// TIA Portal V20 export
// export: Created 2025-12-01T14:57:44.9159736Z, ExportSetting None, DisplayName Totally Integrated Automation Portal, DisplayVersion V20 Update 3, DisplayName TIA Portal Openness, DisplayVersion V20 Update 3, DisplayName TIA Portal Version Control Interface, DisplayVersion V20 Update 3, DisplayName STEP 7 Professional, DisplayVersion V20 Update 3, DisplayName STEP 7 Safety, DisplayVersion V20 Update 2, DisplayName WinCC Basic/Comfort/Advanced, DisplayVersion V20 Update 3, DisplayName WinCC Professional, DisplayVersion V20 Update 3, DisplayName WinCC Unified, DisplayVersion V20 Update 3
FUNCTION "FC780_Evento_RUET" : Void   // FC780, LAD
{ S7_Optimized_Access := 'FALSE' }
// stored: AutoNumber false, SetENOAutomatically false
   VAR_INPUT
      mensaje : Int;   // indice del array que estamos extrayendo
   END_VAR
   VAR_TEMP
      Existe_ruta : Bool;
      retval : Int;
      pos_SSCC : UInt;
      cero : Byte;
      destinos : Array[0..9] of UInt;
      registro_etiqueta : "ROUT_Reg_Etiqueta";
      orden_desvio : Byte;
      desvio_bits AT orden_desvio : Array[1..8] of Bool;
      posicion : Int;
      pos_ruta : Int;
      posicion_mesa : Int;
      posicion_db : Int;
      desvio : Int;
      scanner : UInt;
      bit_ini : Int;
      n_bits : Int;
      contador_aux : Int;
      contador : Int;
      posicion_BBDD : UInt;
      pos_DB : UInt;
      posicion_libre_BBDD : UInt;
      cola : UInt;
      mi_siguiente : UInt;
      dato_actual_cola : UInt;
   END_VAR
BEGIN

REGION Network 1 (SCL): INICIALIZACIONES
   REGION inicializacion

       // inicializamos las variables
       // 
       #cero := 0;
       #retval := FILL(BVAL := #cero, BLK => #registro_etiqueta); // el registro de la etiqueta temporal
       #retval := FILL(BVAL := #cero, BLK => #destinos); // los datos temporales de los destinos
       #orden_desvio := 0;
       #Existe_ruta := false;
       #pos_SSCC := 0;

   END_REGION
END_REGION

REGION Network 2 (SCL): RECOJO Y CONVIERTO EL VALOR DE LA EITQUETA
   // buscamos donde empieza el SSCC en el mensaje y lo convertimos
   // 
   #pos_SSCC := FIND(IN1 := "DB199_eventos_convertidos".evento[#mensaje], IN2 := '[SSCC]');

   STRG_VAL(IN := "DB199_eventos_convertidos".evento[#mensaje],
            FORMAT := 0,
            P := (#pos_SSCC + 6), // +6 por lo que ocupa el atributo ['SSCC]'
            OUT => #registro_etiqueta.CDB);
END_REGION

REGION Network 3 (SCL): EXTRAEMOS DEL MENSAJE LOS DESTINOS

   // miramos si en el mensaje nos han llegado destinos que extraer
   #posicion := FIND(IN1 := "DB199_eventos_convertidos".evento[#mensaje], IN2 := '[DEST]');
   IF #posicion <> 0 THEN    // iniciamos la estracción de las mesas que pertenecen a la ruta
           // si solamente se ejecuta el proceso una vez en el mensaje no es necesario realizar esta operación de sustituir el atributo DEST
       "DB199_eventos_convertidos".evento[#mensaje] := REPLACE(IN1 := "DB199_eventos_convertidos".evento[#mensaje], IN2 := '[dest]', L := 6, P := #posicion);
       #pos_ruta := 0;
       #Existe_ruta := 1;
       // temporalmente ponemos las rutas a cero
       WHILE #Existe_ruta DO
           #posicion := FIND(IN1 := "DB199_eventos_convertidos".evento[#mensaje], IN2 := '[MESA]');
           IF #posicion <> 0 THEN
               STRG_VAL(IN := "DB199_eventos_convertidos".evento[#mensaje],
                        FORMAT := 0,
                        P := (#posicion + 6),
                        OUT => #destinos[#pos_ruta]);
               #pos_ruta += 1; // incrementamos la posición en el array para seguir guardando
               // las mesas ya extraidas, las ponemos en minucula para seguir buscando las siguientes mesas sin eliminar parcialmente el mensaje
               "DB199_eventos_convertidos".evento[#mensaje] := REPLACE(IN1 := "DB199_eventos_convertidos".evento[#mensaje], IN2 := '[mesa]', L := 6, P := #posicion);
           ELSE
               #Existe_ruta := 0;
               EXIT;
           END_IF;
       END_WHILE;
   END_IF;
   // aqui tenemos que incluir la conversión de las mesas el los bits de cruce
END_REGION

REGION Network 4 (SCL): generamos los bits de cruce
   REGION generar_bits_cruce
       #posicion_mesa := 0;
       #posicion_db := 0;

       WHILE #destinos[#posicion_mesa] <> 0 DO
           // Statement section WHILE

           WHILE (("DB913_Router_DestinoDesvio".DestinoDesvios[#posicion_db].Destino <> 0) AND (#posicion_db <= "ROUT_Max_Destinos")) DO
               IF (#destinos[#posicion_mesa] = "DB913_Router_DestinoDesvio".DestinoDesvios[#posicion_db].Destino) THEN
                   // si coincide la mesa con uno de los destinos
                   #desvio := 0;
                   WHILE (("DB913_Router_DestinoDesvio".DestinoDesvios[#posicion_db].Desvios[#desvio].SCR <> 0) AND (#desvio <= "ROUT_Max_Destinos")) DO
                       #scanner := "DB913_Router_DestinoDesvio".DestinoDesvios[#posicion_db].Desvios[#desvio].SCR;
                       #orden_desvio := "DB913_Router_DestinoDesvio".DestinoDesvios[#posicion_db].Desvios[#desvio].Bits;
                       #bit_ini := "DB912_Tipo_Scanner_Router".SCANNER[#scanner].Bit_Ini_Ordenes;
                       #n_bits := "DB912_Tipo_Scanner_Router".SCANNER[#scanner].N_Bits_Orden;

                       // aqui mediante un for vamos escribiendo los bits donde corresponden
                       #contador_aux := 1;
                       FOR #contador := #bit_ini TO (#bit_ini + #n_bits - 1) DO
                           #registro_etiqueta.BIT_Orden[#contador] := #desvio_bits[#contador_aux];
                           #contador_aux += 1;

                       END_FOR;
                       #desvio += 1; // nos desplazamos el siguiente desvio
                   END_WHILE;

               END_IF;
               #posicion_db += 1; //nos desplazamos hasta el siguiente destino
           END_WHILE;
           #posicion_mesa += 1; // nos desplazamos a la siguiente mesa destino de la ruta
           #posicion_db := 0; // inicializamos a cero la busqueda dentro del DB de destinos

       END_WHILE;

   END_REGION
END_REGION

REGION Network 5 (SCL)
   // ahora que tenemos todos los datos, tenemos que guardarlos.
   // miramos si la etiqueta ya está dada de alta en la BBDD
   // 

   "FC715_Router_BuscarEtiqueta_Lint"(Etiqueta := #registro_etiqueta.CDB,
                                      Posicion_BBDD => #posicion_BBDD);

   // si nos da una posición dentro de la BBDD lo unico que tenemos que hacer es sobreescribir el registo
   // si nos da cero, es que no existe y hay que crearla en la primera posición que esté libre
   // 

   REGION escribir_etiqueta_en_BBDD
       // la etiqueta existe
       // 

       REGION existe_etiqueta
           IF #posicion_BBDD <> 0 THEN
               // en función de la posición que nos devuelva, tenemos que ir a un DB diferente
               // 
               REGION elegir_db_busqueda
                   CASE #posicion_BBDD OF
                       1..1000:
                           #pos_DB := #posicion_BBDD;
                           "DB201_RegEtiquetas_0001_1000".Reg_Etiqueta[#pos_DB].BIT_Orden := #registro_etiqueta.BIT_Orden;
                       1001..2000:
                           #pos_DB := #posicion_BBDD - 1000;
                           "DB202_RegEtiquetas_1001_2000".Reg_Etiqueta[#pos_DB].BIT_Orden := #registro_etiqueta.BIT_Orden;

                       2001..3000:
                           #pos_DB := #posicion_BBDD - 2000;
                           "DB203_RegEtiquetas_2001_3000".Reg_Etiqueta[#pos_DB].BIT_Orden := #registro_etiqueta.BIT_Orden;
                       3001..4000:
                           #pos_DB := #posicion_BBDD - 3000;
                           "DB204_RegEtiquetas_3001_4000".Reg_Etiqueta[#pos_DB].BIT_Orden := #registro_etiqueta.BIT_Orden;
                       ELSE
                           #posicion_BBDD := 0;
                           RETURN;
                   END_CASE;
               END_REGION


               ;
           END_IF;
       END_REGION


       REGION no_existe_etiqueta
           IF #posicion_BBDD = 0 THEN
               // 
               // buscamos la primera posición libre dentro de la BBDD que es lo mismo que buscar la primera etiqueta 0
               // 
               "FC715_Router_BuscarEtiqueta_Lint"(Etiqueta := -1,
                                                  Posicion_BBDD => #posicion_libre_BBDD);

               // si la posicion que devuelve es -1 no hay sitio en la BBDD y no se puede crear la etiqueta.
               // 

               IF #posicion_libre_BBDD = -1 THEN
                   "FC818_Mensaje_BBDD_Routing_Llena"(Etiqueta:=#registro_etiqueta.CDB,
                                                      Envio_JDT2:=(NOT("ROUT_X_CONEX_JDT1")));
                   RETURN;

               END_IF;


               // tambien vamos a extraer el valor de la primera etiqueta de la cola para mantener la coherencia de las colas
               // 
               #cola := #registro_etiqueta.CDB MOD "ROUT_N_Colas";
               #dato_actual_cola := "DB212_Cola_Activa".Cola[#cola];
               "DB212_Cola_Activa".Cola[#cola] := #posicion_libre_BBDD;

               IF #dato_actual_cola <> 0 THEN
                   // no es la primera etiqueta de la cola
                   // ahora yo seré el primero de la cola, y el indicado por el valor dato actual será mi siguiente
                   // y yo su anterior
                   // 



                   CASE #dato_actual_cola OF
                       1..1000:
                           #pos_DB := #dato_actual_cola;
                           "DB201_RegEtiquetas_0001_1000".Reg_Etiqueta[#pos_DB].Anterior := #posicion_libre_BBDD;

                       1001..2000:
                           #pos_DB := #dato_actual_cola - 1000;
                           "DB202_RegEtiquetas_1001_2000".Reg_Etiqueta[#pos_DB].Anterior := #posicion_libre_BBDD;

                       2001..3000:
                           #pos_DB := #dato_actual_cola - 2000;
                           "DB203_RegEtiquetas_2001_3000".Reg_Etiqueta[#pos_DB].Anterior := #posicion_libre_BBDD;
                       3001..4000:
                           #pos_DB := #dato_actual_cola - 3000;
                           "DB204_RegEtiquetas_3001_4000".Reg_Etiqueta[#pos_DB].Anterior := #posicion_libre_BBDD;

                           RETURN;
                   END_CASE;

                   #registro_etiqueta.Posterior := #dato_actual_cola;
               END_IF;

               REGION elegir_db_busqueda
                   CASE #posicion_libre_BBDD OF
                       1..1000:
                           #pos_DB := #posicion_libre_BBDD;
                           "DB201_RegEtiquetas_0001_1000".Reg_Etiqueta[#pos_DB] := #registro_etiqueta;

                       1001..2000:
                           #pos_DB := #posicion_libre_BBDD - 1000;
                           "DB202_RegEtiquetas_1001_2000".Reg_Etiqueta[#pos_DB] := #registro_etiqueta;

                       2001..3000:
                           #pos_DB := #posicion_libre_BBDD - 2000;
                           "DB203_RegEtiquetas_2001_3000".Reg_Etiqueta[#pos_DB] := #registro_etiqueta;
                       3001..4000:
                           #pos_DB := #posicion_libre_BBDD - 3000;
                           "DB204_RegEtiquetas_3001_4000".Reg_Etiqueta[#pos_DB] := #registro_etiqueta;

                           RETURN;
                   END_CASE;
               END_REGION

           END_IF;
       END_REGION

   END_REGION

   #retval := FILL(BVAL := #registro_etiqueta, BLK => "DB209_Reg_Etquetas_Esp_Activa".Reg_Etiqueta[5]);
END_REGION
END_FUNCTION
